Fanuc KAREL source: kt00049.KL

-- PROVISIONAL review KL for V1013-1; original PC SHA256 7f21acbac08ef576589d9baf3d85900afb7b01365d777da2c1719b2cddafaf1a
-- Incomplete behavior may be omitted. Consult companion uncertainty JSON. Do not deploy.
PROGRAM KT00049
%NOLOCKGROUP
VAR
  I2 : INTEGER
  OUT : INTEGER
-- UNRESOLVED_DECL Y1 type=002018
BEGIN
  -- UNRESOLVED_PC offsets 5-19; opcodes 2E,22,9D,33,B2
  -- UNRESOLVED_PC offsets 24-35; opcodes 2E,23
  -- UNRESOLVED_PC offsets 40-62; opcodes 22,9D,33,B1,21,53,23
  -- UNRESOLVED_PC offsets 67-71; opcodes 7F
END KT00049
